PROGRAM PRG_Task3
VAR
END_VAR

F_ConsumeTime(4000);

END_PROGRAM

(* stored: Version 1.1.0.1, ProductVersion 3.1.4026.18
   POU PRG_Task3: Id {85c175b3-461d-47f0-bac3-341d32a49887}, SpecialFunc None *)
